{attribute 'qualified_only'}


VAR_GLOBAL
	StatusWord_Bits :  Ds402_SW;
	DirUp : BOOL;
	ProfParams : Ds402_Params;

END_VAR

(* stored: Version 1.1.0.1, ProductVersion 3.1.4024.6
   GVL Ds402: Id {6f396431-a803-4521-86de-c14f520c6927} *)
